// TIA Portal V20 export
DATA_BLOCK "BK05"   // DB307
// stored: MemoryReserve 100
   VAR
      "X10-1.ANODE MAIN P&P1 Z-AXIS LIMIT SENSOR(-)" : Bool := TRUE;
      "X11-1.ANODE MAIN P&P1 Z-AXIS LIMIT SENSOR(+)" : Bool := TRUE;
      "X12-1.ANODE MAIN P&P1 Y-AXIS LIMIT SENSOR(-)" : Bool := TRUE;
      "X13-1.ANODE MAIN P&P1 Y-AXIS LIMIT SENSOR(+)" : Bool := TRUE;
      "X14-1.SPARE" : Bool := FALSE;
      "X15-1.ANODE MAIN P&P1 DETECT SENSOR" : Bool := FALSE;
      "X16-1.ANODE MAIN P&P1 ROTARY CCW" : Bool := FALSE;
      "X17-1.ANODE MAIN P&P1 PRESSURE SWITCH" : Bool := FALSE;
      "X10-2.ANODE MAIN P&P1 Z-AXIS HOME SENSOR" : Bool := TRUE;
      "X11-2.SPARE" : Bool := FALSE;
      "X12-2.ANODE MAIN P&P1 Y-AXIS HOME SENSOR" : Bool := TRUE;
      "X13-2.SPARE" : Bool := FALSE;
      "X14-2.SPARE" : Bool := FALSE;
      "X15-2.SPARE" : Bool := FALSE;
      "X16-2.ANODE MAIN P&P1 ROTARY CW" : Bool := TRUE;
      "X17-2.SPARE" : Bool := FALSE;
   END_VAR
BEGIN
END_DATA_BLOCK
